(* PLC project tni_clock, Dassault Systèmes ControlBuild 2019 FD01 Beta 2 *)
(* stored: creationDateTime 2018-09-12T11:57:14-01:00 *)

CONFIGURATION tni_clock
  VAR_GLOBAL
    B1 AT 5 : BOOL := false;
    B2 AT 6 : BOOL := false;
    B3 AT 7 : BOOL := false;
    B4 AT 8 : BOOL := false;
    depth AT 523 : INT := 0;
    environment/depth AT 523 : INT := 0;
    environment/B1 AT 5 : BOOL := false;
    environment/B2 AT 6 : BOOL := false;
    environment/B3 AT 7 : BOOL := false;
    environment/B4 AT 8 : BOOL := false;
    environment/pressure AT 524 : INT := 0;
    environment/tick AT 9 : BOOL := false;
    environment/hydrostaticPressure AT 17 : REAL := 0.0;
    environment/absolutePressure AT 18 : REAL := 0.0;
    controller/pressure AT 524 : INT := 0;
    controller/tick AT 9 : BOOL := false;
    controller/B1 AT 5 : BOOL := false;
    controller/B2 AT 6 : BOOL := false;
    controller/B3 AT 7 : BOOL := false;
    controller/B4 AT 8 : BOOL := false;
    controller/displayValue AT 525 : ARRAY[1..8] OF BYTE := [8(0)];
    controller/stepMotorSecond AT 10 : BOOL := false;
    controller/stepMotorMinute AT 11 : BOOL := false;
    controller/stepMotorHour AT 12 : BOOL := false;
    controller/switchOnLight AT 13 : BOOL := false;
    controller/timeManagement/tick AT 9 : BOOL := false;
    controller/timeManagement/B1 AT 5 : BOOL := false;
    controller/timeManagement/B2 AT 6 : BOOL := false;
    controller/timeManagement/B3 AT 7 : BOOL := false;
    controller/timeManagement/B4 AT 8 : BOOL := false;
    controller/timeManagement/stepMotorSecond AT 10 : BOOL := false;
    controller/timeManagement/stepMotorMinute AT 11 : BOOL := false;
    controller/timeManagement/stepMotorHour AT 12 : BOOL := false;
    controller/timeManagement/hh AT 535 : SINT := 0;
    controller/timeManagement/mn AT 536 : SINT := 0;
    controller/timeManagement/sec AT 537 : SINT := 0;
    controller/timeManagement/tickCount AT 19 : REAL := 0.0;
    controller/timeManagement/adjustMode AT 538 : INT := 0;
    controller/displayManagement/hh AT 535 : SINT := 0;
    controller/displayManagement/mn AT 536 : SINT := 0;
    controller/displayManagement/sec AT 537 : SINT := 0;
    controller/displayManagement/tick AT 9 : BOOL := false;
    controller/displayManagement/pressure AT 524 : INT := 0;
    controller/displayManagement/B1 AT 5 : BOOL := false;
    controller/displayManagement/B2 AT 6 : BOOL := false;
    controller/displayManagement/B3 AT 7 : BOOL := false;
    controller/displayManagement/B4 AT 8 : BOOL := false;
    controller/displayManagement/displayValue AT 525 : ARRAY[1..8] OF BYTE := [8(0)];
    controller/displayManagement/switchOnLight AT 13 : BOOL := false;
    controller/displayManagement/displayTime AT 20 : REAL := 0.0;
    controller/displayManagement/lampSwitchOnTime AT 21 : REAL := 0.0;
    controller/displayManagement/pulseTime AT 540 : DINT := 10;
    LCD/displayValue AT 525 : ARRAY[1..8] OF BYTE := [8(0)];
    LCD/displayString AT 53 : STRING(8) := '';
    LCD/i AT 541 : SINT := 0;
    motors/stepMotorSecond AT 10 : BOOL := false;
    motors/stepMotorMinute AT 11 : BOOL := false;
    motors/stepMotorHour AT 12 : BOOL := false;
    motors/hourHand AT 542 : INT := 0;
    motors/minuteHand AT 543 : INT := 0;
    motors/secondHand AT 544 : INT := 0;
    light/switchOnLight AT 13 : BOOL := false;
  END_VAR
END_CONFIGURATION
